// TIA Portal V16 export
// export: Created 2021-05-25T16:14:42.3691804Z, ExportSetting WithDefaults, DisplayName Totally Integrated Automation Portal, DisplayVersion V16, DisplayName TIA Portal Version Control Interface, DisplayVersion V16, DisplayName TIA Portal Openness, DisplayVersion V16, DisplayName STEP 7 Professional, DisplayVersion V16, DisplayName STEP 7 Safety, DisplayVersion V16, DisplayName WinCC Unified SCADA Engineering System, DisplayVersion V16
DATA_BLOCK "dbMotors"   // DB33
{ S7_Optimized_Access := 'TRUE'; DB_Accessible_From_OPC_UA := 'FALSE' }
VERSION : 0.1
// stored: AutoNumber false, DBAccessibleFromOPCUA false, IsOnlyStoredInLoadMemory false, IsRetainMemResEnabled false, IsWriteProtectedInAS false, MemoryReserve 100
   VAR
      VKLOP_M_TRACNEGA_TRANS_NOGIC : "udtMotor";
      M1_ZADAJ_DESNO : "udtMotor";
      M2_SPREDAJ_DESNO : "udtMotor";
      M1_ZADAJ_LEVO : "udtMotor";
      M2_SPREDAJ_LEVO : "udtMotor";
      VKLOP_VIBRATORJA : "udtMotor";
      VKLOP_M_TRAKA_VIJACNIKA : "udtMotor";
   END_VAR
BEGIN
END_DATA_BLOCK
